(* PLC project Unnamed, Unknown Unnamed 1 *)
(* stored: creationDateTime 2026-04-26T22:09:28, modificationDateTime 2026-04-26T22:09:28 *)

FUNCTION_BLOCK BOOL_ON_WORD
  VAR_INPUT
    B_IN0 : BOOL;
    B_IN1 : BOOL;
    B_IN2 : BOOL;
    B_IN3 : BOOL;
    B_IN4 : BOOL;
    B_IN5 : BOOL;
    B_IN6 : BOOL;
    B_IN7 : BOOL;
    B_IN8 : BOOL;
    B_IN9 : BOOL;
    B_IN10 : BOOL;
    B_IN11 : BOOL;
    B_IN12 : BOOL;
    B_IN13 : BOOL;
    B_IN14 : BOOL;
    B_IN15 : BOOL;
  END_VAR
  VAR_OUTPUT
    WORD_OUT : WORD;
  END_VAR

            WORD_OUT := 0;
IF B_IN0  THEN WORD_OUT := WORD_OUT OR 16#0001; END_IF;
IF B_IN1  THEN WORD_OUT := WORD_OUT OR 16#0002; END_IF;
IF B_IN2  THEN WORD_OUT := WORD_OUT OR 16#0004; END_IF;
IF B_IN3  THEN WORD_OUT := WORD_OUT OR 16#0008; END_IF;
IF B_IN4  THEN WORD_OUT := WORD_OUT OR 16#0010; END_IF;
IF B_IN5  THEN WORD_OUT := WORD_OUT OR 16#0020; END_IF;
IF B_IN6  THEN WORD_OUT := WORD_OUT OR 16#0040; END_IF;
IF B_IN7  THEN WORD_OUT := WORD_OUT OR 16#0080; END_IF;
IF B_IN8  THEN WORD_OUT := WORD_OUT OR 16#0100; END_IF;
IF B_IN9  THEN WORD_OUT := WORD_OUT OR 16#0200; END_IF;
IF B_IN10 THEN WORD_OUT := WORD_OUT OR 16#0400; END_IF;
IF B_IN11 THEN WORD_OUT := WORD_OUT OR 16#0800; END_IF;
IF B_IN12 THEN WORD_OUT := WORD_OUT OR 16#1000; END_IF;
IF B_IN13 THEN WORD_OUT := WORD_OUT OR 16#2000; END_IF;
IF B_IN14 THEN WORD_OUT := WORD_OUT OR 16#4000; END_IF;
IF B_IN15 THEN WORD_OUT := WORD_OUT OR 16#8000; END_IF;
          
END_FUNCTION_BLOCK

FUNCTION_BLOCK CAN_INTERFACE
  VAR_INPUT
    ID_FILTER : INT := 300;
    ID_STATE : INT := 310;
    STATE_PERIOD : INT := 500;
    INPUT_ADDRESS : INT := 0;
    NUM_OF_INPUT : INT := 1;
    OUTPUT_ADDRESS : INT := 2;
    NUM_OF_OUTPUT : INT := 1;
  END_VAR
  VAR_OUTPUT
    ERR : BOOL;
  END_VAR
  VAR
    hasBeenInitialized : BOOL := 0;
  END_VAR

            {{
CAN_INTERFACE_VARS vars;
vars.ID_FILTER = &data__->ID_FILTER.value;
vars.ID_STATE = &data__->ID_STATE.value;
vars.STATE_PERIOD = &data__->STATE_PERIOD.value;
vars.INPUT_ADDRESS = &data__->INPUT_ADDRESS.value;
vars.NUM_OF_INPUT = &data__->NUM_OF_INPUT.value;
vars.OUTPUT_ADDRESS = &data__->OUTPUT_ADDRESS.value;
vars.NUM_OF_OUTPUT = &data__->NUM_OF_OUTPUT.value;
vars.ERR = &data__->ERR.value;
}}
if hasBeenInitialized = False then
{{
can_interface_setup(&vars);
}}
hasBeenInitialized := True;
end_if;
{{
can_interface_loop(&vars);
}}
          
END_FUNCTION_BLOCK

FUNCTION_BLOCK WORD_ON_BOOL
  VAR_INPUT
    WORD_IN : WORD;
  END_VAR
  VAR_OUTPUT
    B_OUT0 : BOOL;
    B_OUT1 : BOOL;
    B_OUT2 : BOOL;
    B_OUT3 : BOOL;
    B_OUT4 : BOOL;
    B_OUT5 : BOOL;
    B_OUT6 : BOOL;
    B_OUT7 : BOOL;
    B_OUT8 : BOOL;
    B_OUT9 : BOOL;
    B_OUT10 : BOOL;
    B_OUT11 : BOOL;
    B_OUT12 : BOOL;
    B_OUT13 : BOOL;
    B_OUT14 : BOOL;
    B_OUT15 : BOOL;
  END_VAR

            B_OUT0  := (WORD_IN AND 16#0001) <> 0;
B_OUT1  := (WORD_IN AND 16#0002) <> 0;
B_OUT2  := (WORD_IN AND 16#0004) <> 0;
B_OUT3  := (WORD_IN AND 16#0008) <> 0;
B_OUT4  := (WORD_IN AND 16#0010) <> 0;
B_OUT5  := (WORD_IN AND 16#0020) <> 0;
B_OUT6  := (WORD_IN AND 16#0040) <> 0;
B_OUT7  := (WORD_IN AND 16#0080) <> 0;
B_OUT8  := (WORD_IN AND 16#0100) <> 0;
B_OUT9  := (WORD_IN AND 16#0200) <> 0;
B_OUT10 := (WORD_IN AND 16#0400) <> 0;
B_OUT11 := (WORD_IN AND 16#0800) <> 0;
B_OUT12 := (WORD_IN AND 16#1000) <> 0;
B_OUT13 := (WORD_IN AND 16#2000) <> 0;
B_OUT14 := (WORD_IN AND 16#4000) <> 0;
B_OUT15 := (WORD_IN AND 16#8000) <> 0;
          
END_FUNCTION_BLOCK

PROGRAM main
  VAR
    BTN_ON_1 AT %IX0.3 : BOOL;
    BTN_ON_2 AT %IX0.5 : BOOL;
    K1 AT %QX0.0 : BOOL;
    K2 AT %QX0.1 : BOOL;
    BTN_OFF_1 AT %IX0.4 : BOOL;
    BTN_OFF_2 AT %IX0.6 : BOOL;
    CMD_WORD AT %MW0 : WORD;
    CYRCLE_STATE AT %MW1 : WORD := 0;
    CAN_STATE AT %MW2 : WORD;
  END_VAR
  VAR
    CAN_ERR : BOOL;
    K1_CAN_ON : BOOL;
    K2_CAN_ON : BOOL;
    K1_CAN_OFF : BOOL;
    K2_CAN_OFF : BOOL;
    BTN_ON_1_TMP : BOOL;
    BTN_ON_2_TMP : BOOL;
    BTN_OFF_1_TMP : BOOL;
    BTN_OFF_2_TMP : BOOL;
    TON0_TMP_ON : BOOL;
    TON1_TMP_ON : BOOL;
    TON2_TMP_ON : BOOL;
    TON3_TMP_ON : BOOL;
    CYCLE_RUN : BOOL;
    CYCLE_RUN_SET : BOOL;
    CMD_1 : BOOL;
    CMD_2 : BOOL;
    CMD_3 : BOOL;
    CMD_4 : BOOL;
    TON0 : TON;
    TON1 : TON;
    TON2 : TON;
    TON3 : TON;
    TON4 : TON;
    CAN_INTERFACE0 : CAN_INTERFACE;
    BOOL_ON_WORD0 : BOOL_ON_WORD;
  END_VAR
  VAR  (* added by the conversion: wires and edge detectors of the diagram *)
    _MOVE3435397_ENO : BOOL;
    _MOVE3435397_OUT : WORD;
    _MOVE8007104_ENO : BOOL;
    _MOVE8007104_OUT : WORD;
    _MOVE656876_ENO : BOOL;
    _MOVE656876_OUT : WORD;
    _MOVE4683258_ENO : BOOL;
    _MOVE4683258_OUT : WORD;
    _MOVE6517896_ENO : BOOL;
    _MOVE6517896_OUT : WORD;
    R_TRIG1 : R_TRIG;
    R_TRIG2 : R_TRIG;
    R_TRIG3 : R_TRIG;
    R_TRIG4 : R_TRIG;
    R_TRIG5 : R_TRIG;
    R_TRIG6 : R_TRIG;
  END_VAR

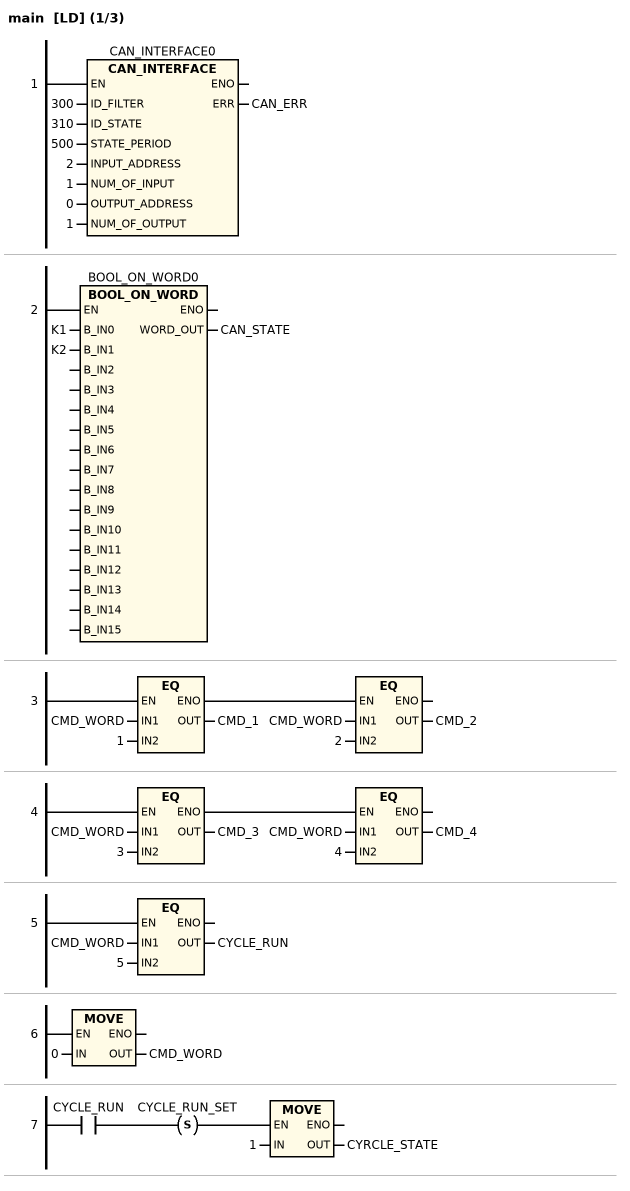
(* LD diagram, written out as Structured Text *)
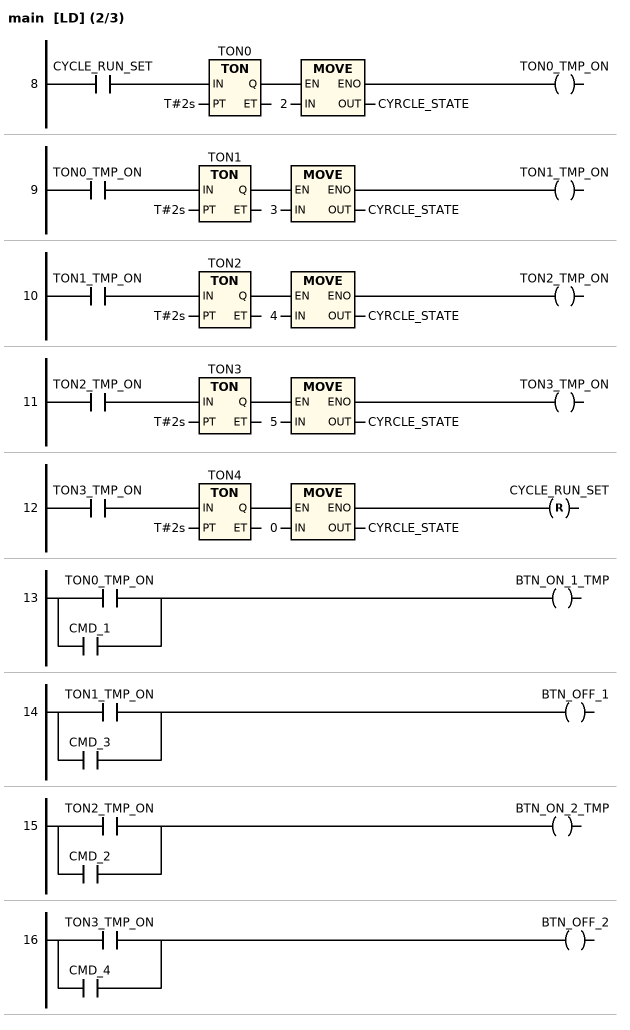
IF CYCLE_RUN THEN CYCLE_RUN_SET := TRUE; END_IF;
TON0(IN := CYCLE_RUN_SET, PT := T#2s);
_MOVE3435397_OUT := MOVE(EN := TON0.Q, IN := 2, ENO => _MOVE3435397_ENO);
TON0_TMP_ON := _MOVE3435397_ENO;
TON1(IN := TON0_TMP_ON, PT := T#2s);
_MOVE8007104_OUT := MOVE(EN := TON1.Q, IN := 3, ENO => _MOVE8007104_ENO);
TON1_TMP_ON := _MOVE8007104_ENO;
TON2(IN := TON1_TMP_ON, PT := T#2s);
_MOVE656876_OUT := MOVE(EN := TON2.Q, IN := 4, ENO => _MOVE656876_ENO);
TON2_TMP_ON := _MOVE656876_ENO;
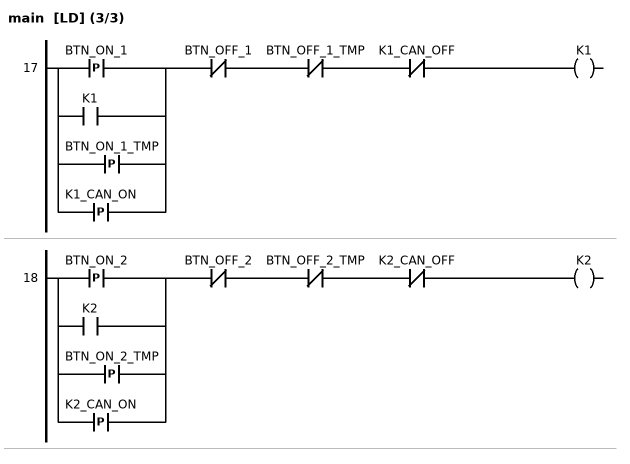
TON3(IN := TON2_TMP_ON, PT := T#2s);
_MOVE4683258_OUT := MOVE(EN := TON3.Q, IN := 5, ENO => _MOVE4683258_ENO);
TON3_TMP_ON := _MOVE4683258_ENO;
TON4(IN := TON3_TMP_ON, PT := T#2s);
_MOVE6517896_OUT := MOVE(EN := TON4.Q, IN := 0, ENO => _MOVE6517896_ENO);
IF _MOVE6517896_ENO THEN CYCLE_RUN_SET := FALSE; END_IF;
BTN_ON_1_TMP := TON0_TMP_ON OR CMD_1;
BTN_OFF_1 := TON1_TMP_ON OR CMD_3;
BTN_ON_2_TMP := TON2_TMP_ON OR CMD_2;
BTN_OFF_2 := TON3_TMP_ON OR CMD_4;
R_TRIG1(CLK := BTN_ON_1);
R_TRIG2(CLK := BTN_ON_1_TMP);
R_TRIG3(CLK := K1_CAN_ON);
K1 := (R_TRIG1.Q OR K1 OR R_TRIG2.Q OR R_TRIG3.Q) AND NOT BTN_OFF_1 AND NOT BTN_OFF_1_TMP AND NOT K1_CAN_OFF;
R_TRIG4(CLK := BTN_ON_2);
R_TRIG5(CLK := BTN_ON_2_TMP);
R_TRIG6(CLK := K2_CAN_ON);
K2 := (R_TRIG4.Q OR K2 OR R_TRIG5.Q OR R_TRIG6.Q) AND NOT BTN_OFF_2 AND NOT BTN_OFF_2_TMP AND NOT K2_CAN_OFF;
CAN_INTERFACE0(ID_FILTER := 300, ID_STATE := 310, STATE_PERIOD := 500, INPUT_ADDRESS := 2, NUM_OF_INPUT := 1, OUTPUT_ADDRESS := 0, NUM_OF_OUTPUT := 1);
CAN_ERR := CAN_INTERFACE0.ERR;
BOOL_ON_WORD0(B_IN0 := K1, B_IN1 := K2);
CAN_STATE := BOOL_ON_WORD0.WORD_OUT;
CMD_1 := CMD_WORD = 1;
CMD_2 := CMD_WORD = 2;
CMD_3 := CMD_WORD = 3;
CMD_4 := CMD_WORD = 4;
CYCLE_RUN := CMD_WORD = 5;
CMD_WORD := 0;
IF CYCLE_RUN THEN CYRCLE_STATE := 1; END_IF;
IF _MOVE3435397_ENO THEN CYRCLE_STATE := _MOVE3435397_OUT; END_IF;
IF _MOVE8007104_ENO THEN CYRCLE_STATE := _MOVE8007104_OUT; END_IF;
IF _MOVE656876_ENO THEN CYRCLE_STATE := _MOVE656876_OUT; END_IF;
IF _MOVE4683258_ENO THEN CYRCLE_STATE := _MOVE4683258_OUT; END_IF;
IF _MOVE6517896_ENO THEN CYRCLE_STATE := _MOVE6517896_OUT; END_IF;
END_PROGRAM

CONFIGURATION Config0
  RESOURCE Res0 ON PLC
    TASK task0(INTERVAL := T#20ms, PRIORITY := 1);
    PROGRAM instance0 WITH task0 : main;
  END_RESOURCE
END_CONFIGURATION
